// TIA Portal V17 export
// export: Created 2025-03-10T13:11:40.6014181Z, ExportSetting WithDefaults, DisplayName Totally Integrated Automation Portal, DisplayVersion V17 Update 8, DisplayName TIA Portal Openness, DisplayVersion V17 Update 8, DisplayName TIA Portal Version Control Interface, DisplayVersion V17, DisplayName SINAMICS Startdrive Advanced, DisplayVersion V17 SP2, DisplayName SINAMICS Startdrive G110M, G120, G120C, G120D, G120P, G115D, DisplayVersion V17 SP2, DisplayName SINAMICS Startdrive G130, G150, S120, S150, SINAMICS MV, S210, DisplayVersion V17 SP2, DisplayName STEP 7 Professional, DisplayVersion V17 Update 8, DisplayName SINUMERIK ONE STEP 7 Toolbox, DisplayVersion V17 Update 12, DisplayName SINUMERIK 840D sl STEP 7 Toolbox, DisplayVersion V17 Update 12, DisplayName STEP 7 Safety, DisplayVersion V17 Update 6, DisplayName WinCC Advanced, DisplayVersion V17 Update 8
FUNCTION "FC7213_CYCLE_TIMES_CLADDING" : Void   // FC7213, LAD
TITLE = FC CYCLE TIMES
{ S7_Optimized_Access := 'FALSE' }
AUTHOR : ETXETAR
VERSION : 1.0
// stored: AutoNumber false, IsIECCheckEnabled false, SetENOAutomatically false, UDAEnableTagReadback false
   VAR_TEMP
      CYCLE_TIME : Int;
      TIMER_INT : Int;
      PART_CYCLE_TIME : Int;
   END_VAR
   VAR_TEMP   // added for the SCL form of the ladder/FBD networks
      _w1 : Bool;
      _w2 : Bool;
      _w3 : Bool;
      _w4 : Bool;
   END_VAR
BEGIN

REGION Network 1: PART TYPE 1 TO 5
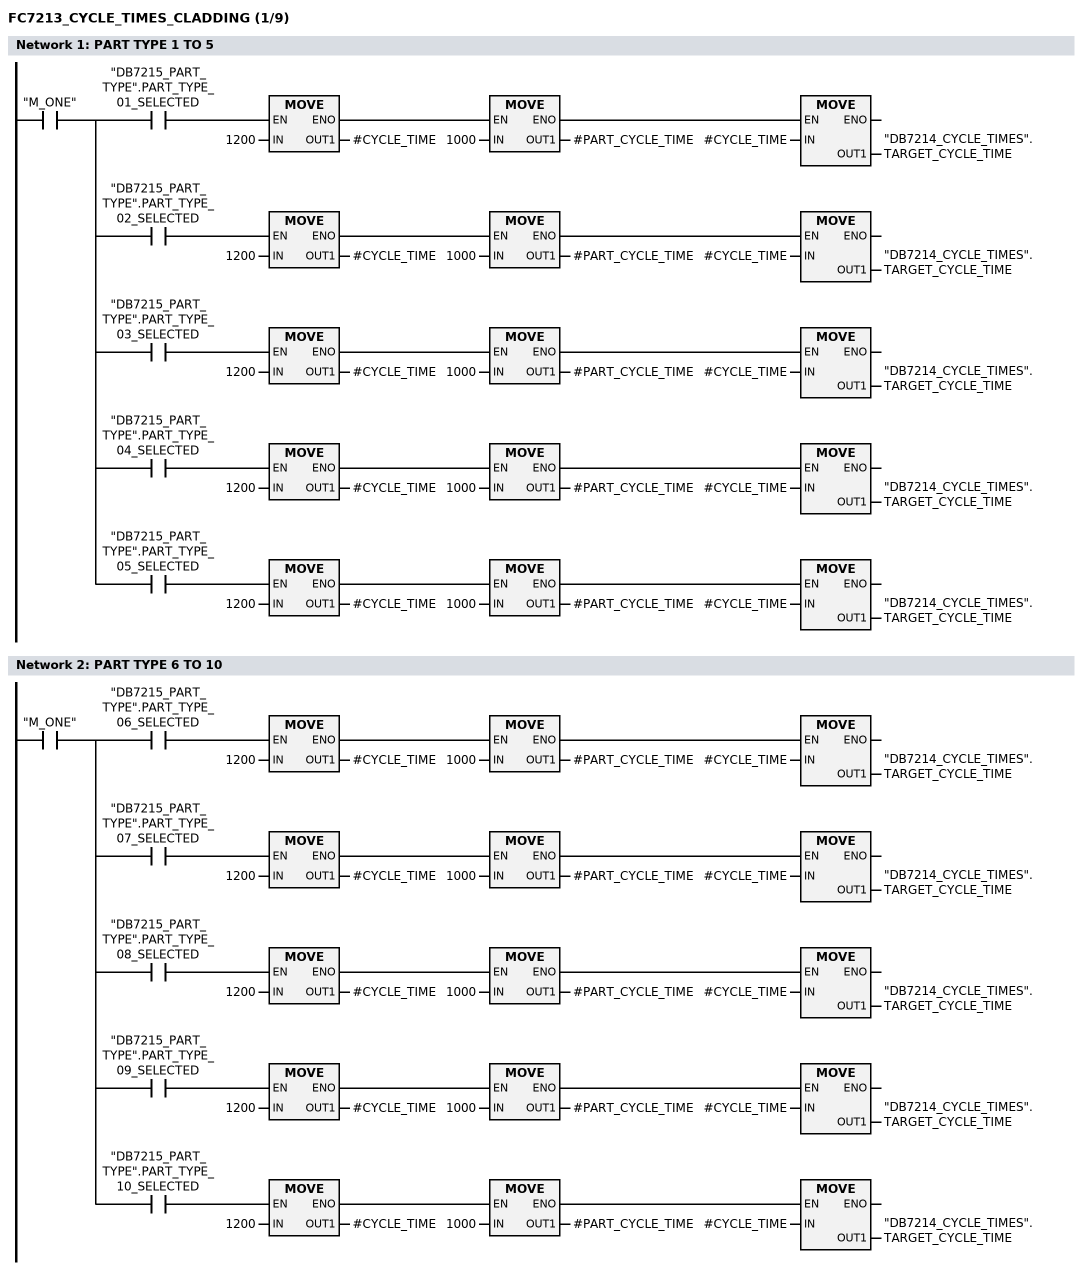
   RUNG wire#powerrail
      Contact( "M_ONE" )
      wire#w1
      Contact( "DB7215_PART_TYPE".PART_TYPE_01_SELECTED )
      { S7_GenerateENO := "TRUE" } Move(in := 1200, out1 => #CYCLE_TIME)
      { S7_GenerateENO := "TRUE" } Move(in := 1000, out1 => #PART_CYCLE_TIME)
      { S7_GenerateENO := "TRUE" } Move(in := #CYCLE_TIME, out1 => "DB7214_CYCLE_TIMES".TARGET_CYCLE_TIME)
   END_RUNG
   RUNG wire#w1
      Contact( "DB7215_PART_TYPE".PART_TYPE_02_SELECTED )
      { S7_GenerateENO := "TRUE" } Move(in := 1200, out1 => #CYCLE_TIME)
      { S7_GenerateENO := "TRUE" } Move(in := 1000, out1 => #PART_CYCLE_TIME)
      { S7_GenerateENO := "TRUE" } Move(in := #CYCLE_TIME, out1 => "DB7214_CYCLE_TIMES".TARGET_CYCLE_TIME)
   END_RUNG
   RUNG wire#w1
      Contact( "DB7215_PART_TYPE".PART_TYPE_03_SELECTED )
      { S7_GenerateENO := "TRUE" } Move(in := 1200, out1 => #CYCLE_TIME)
      { S7_GenerateENO := "TRUE" } Move(in := 1000, out1 => #PART_CYCLE_TIME)
      { S7_GenerateENO := "TRUE" } Move(in := #CYCLE_TIME, out1 => "DB7214_CYCLE_TIMES".TARGET_CYCLE_TIME)
   END_RUNG
   RUNG wire#w1
      Contact( "DB7215_PART_TYPE".PART_TYPE_04_SELECTED )
      { S7_GenerateENO := "TRUE" } Move(in := 1200, out1 => #CYCLE_TIME)
      { S7_GenerateENO := "TRUE" } Move(in := 1000, out1 => #PART_CYCLE_TIME)
      { S7_GenerateENO := "TRUE" } Move(in := #CYCLE_TIME, out1 => "DB7214_CYCLE_TIMES".TARGET_CYCLE_TIME)
   END_RUNG
   RUNG wire#w1
      Contact( "DB7215_PART_TYPE".PART_TYPE_05_SELECTED )
      { S7_GenerateENO := "TRUE" } Move(in := 1200, out1 => #CYCLE_TIME)
      { S7_GenerateENO := "TRUE" } Move(in := 1000, out1 => #PART_CYCLE_TIME)
      { S7_GenerateENO := "TRUE" } Move(in := #CYCLE_TIME, out1 => "DB7214_CYCLE_TIMES".TARGET_CYCLE_TIME)
   END_RUNG
   // the same network as SCL:
   // ENO of a box is taken as its EN; it also drops when the box reports an error
   IF "M_ONE" AND "DB7215_PART_TYPE".PART_TYPE_01_SELECTED THEN
       #CYCLE_TIME := 1200;
       #PART_CYCLE_TIME := 1000;
       "DB7214_CYCLE_TIMES".TARGET_CYCLE_TIME := #CYCLE_TIME;
   END_IF;
   IF "M_ONE" AND "DB7215_PART_TYPE".PART_TYPE_02_SELECTED THEN
       #CYCLE_TIME := 1200;
       #PART_CYCLE_TIME := 1000;
       "DB7214_CYCLE_TIMES".TARGET_CYCLE_TIME := #CYCLE_TIME;
   END_IF;
   IF "M_ONE" AND "DB7215_PART_TYPE".PART_TYPE_03_SELECTED THEN
       #CYCLE_TIME := 1200;
       #PART_CYCLE_TIME := 1000;
       "DB7214_CYCLE_TIMES".TARGET_CYCLE_TIME := #CYCLE_TIME;
   END_IF;
   IF "M_ONE" AND "DB7215_PART_TYPE".PART_TYPE_04_SELECTED THEN
       #CYCLE_TIME := 1200;
       #PART_CYCLE_TIME := 1000;
       "DB7214_CYCLE_TIMES".TARGET_CYCLE_TIME := #CYCLE_TIME;
   END_IF;
   IF "M_ONE" AND "DB7215_PART_TYPE".PART_TYPE_05_SELECTED THEN
       #CYCLE_TIME := 1200;
       #PART_CYCLE_TIME := 1000;
       "DB7214_CYCLE_TIMES".TARGET_CYCLE_TIME := #CYCLE_TIME;
   END_IF;
END_REGION

REGION Network 2: PART TYPE 6 TO 10
   RUNG wire#powerrail
      Contact( "M_ONE" )
      wire#w1
      Contact( "DB7215_PART_TYPE".PART_TYPE_06_SELECTED )
      { S7_GenerateENO := "TRUE" } Move(in := 1200, out1 => #CYCLE_TIME)
      { S7_GenerateENO := "TRUE" } Move(in := 1000, out1 => #PART_CYCLE_TIME)
      { S7_GenerateENO := "TRUE" } Move(in := #CYCLE_TIME, out1 => "DB7214_CYCLE_TIMES".TARGET_CYCLE_TIME)
   END_RUNG
   RUNG wire#w1
      Contact( "DB7215_PART_TYPE".PART_TYPE_07_SELECTED )
      { S7_GenerateENO := "TRUE" } Move(in := 1200, out1 => #CYCLE_TIME)
      { S7_GenerateENO := "TRUE" } Move(in := 1000, out1 => #PART_CYCLE_TIME)
      { S7_GenerateENO := "TRUE" } Move(in := #CYCLE_TIME, out1 => "DB7214_CYCLE_TIMES".TARGET_CYCLE_TIME)
   END_RUNG
   RUNG wire#w1
      Contact( "DB7215_PART_TYPE".PART_TYPE_08_SELECTED )
      { S7_GenerateENO := "TRUE" } Move(in := 1200, out1 => #CYCLE_TIME)
      { S7_GenerateENO := "TRUE" } Move(in := 1000, out1 => #PART_CYCLE_TIME)
      { S7_GenerateENO := "TRUE" } Move(in := #CYCLE_TIME, out1 => "DB7214_CYCLE_TIMES".TARGET_CYCLE_TIME)
   END_RUNG
   RUNG wire#w1
      Contact( "DB7215_PART_TYPE".PART_TYPE_09_SELECTED )
      { S7_GenerateENO := "TRUE" } Move(in := 1200, out1 => #CYCLE_TIME)
      { S7_GenerateENO := "TRUE" } Move(in := 1000, out1 => #PART_CYCLE_TIME)
      { S7_GenerateENO := "TRUE" } Move(in := #CYCLE_TIME, out1 => "DB7214_CYCLE_TIMES".TARGET_CYCLE_TIME)
   END_RUNG
   RUNG wire#w1
      Contact( "DB7215_PART_TYPE".PART_TYPE_10_SELECTED )
      { S7_GenerateENO := "TRUE" } Move(in := 1200, out1 => #CYCLE_TIME)
      { S7_GenerateENO := "TRUE" } Move(in := 1000, out1 => #PART_CYCLE_TIME)
      { S7_GenerateENO := "TRUE" } Move(in := #CYCLE_TIME, out1 => "DB7214_CYCLE_TIMES".TARGET_CYCLE_TIME)
   END_RUNG
   // the same network as SCL:
   // ENO of a box is taken as its EN; it also drops when the box reports an error
   IF "M_ONE" AND "DB7215_PART_TYPE".PART_TYPE_06_SELECTED THEN
       #CYCLE_TIME := 1200;
       #PART_CYCLE_TIME := 1000;
       "DB7214_CYCLE_TIMES".TARGET_CYCLE_TIME := #CYCLE_TIME;
   END_IF;
   IF "M_ONE" AND "DB7215_PART_TYPE".PART_TYPE_07_SELECTED THEN
       #CYCLE_TIME := 1200;
       #PART_CYCLE_TIME := 1000;
       "DB7214_CYCLE_TIMES".TARGET_CYCLE_TIME := #CYCLE_TIME;
   END_IF;
   IF "M_ONE" AND "DB7215_PART_TYPE".PART_TYPE_08_SELECTED THEN
       #CYCLE_TIME := 1200;
       #PART_CYCLE_TIME := 1000;
       "DB7214_CYCLE_TIMES".TARGET_CYCLE_TIME := #CYCLE_TIME;
   END_IF;
   IF "M_ONE" AND "DB7215_PART_TYPE".PART_TYPE_09_SELECTED THEN
       #CYCLE_TIME := 1200;
       #PART_CYCLE_TIME := 1000;
       "DB7214_CYCLE_TIMES".TARGET_CYCLE_TIME := #CYCLE_TIME;
   END_IF;
   IF "M_ONE" AND "DB7215_PART_TYPE".PART_TYPE_10_SELECTED THEN
       #CYCLE_TIME := 1200;
       #PART_CYCLE_TIME := 1000;
       "DB7214_CYCLE_TIMES".TARGET_CYCLE_TIME := #CYCLE_TIME;
   END_IF;
END_REGION

REGION Network 3: PART TYPE 11 TO 15
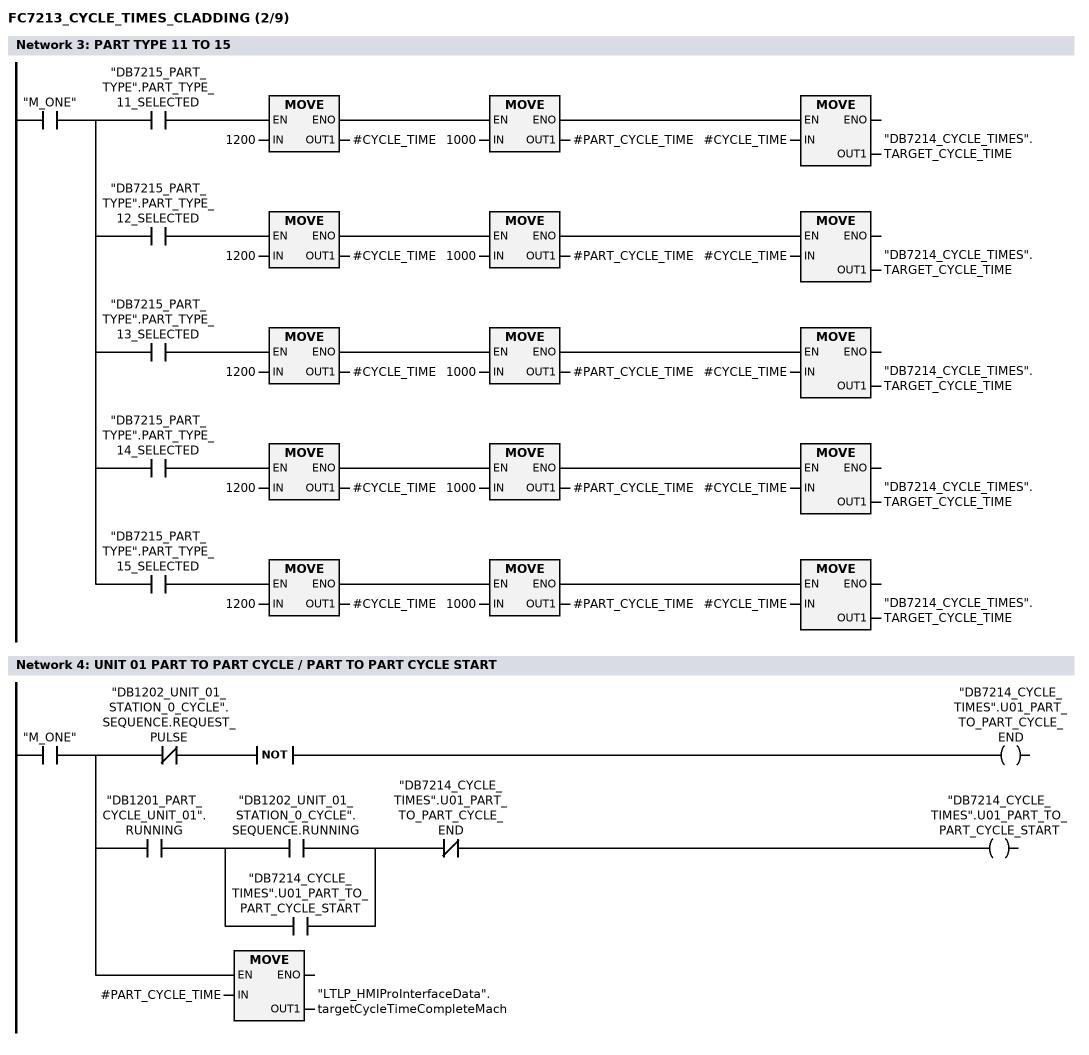
   RUNG wire#powerrail
      Contact( "M_ONE" )
      wire#w1
      Contact( "DB7215_PART_TYPE".PART_TYPE_11_SELECTED )
      { S7_GenerateENO := "TRUE" } Move(in := 1200, out1 => #CYCLE_TIME)
      { S7_GenerateENO := "TRUE" } Move(in := 1000, out1 => #PART_CYCLE_TIME)
      { S7_GenerateENO := "TRUE" } Move(in := #CYCLE_TIME, out1 => "DB7214_CYCLE_TIMES".TARGET_CYCLE_TIME)
   END_RUNG
   RUNG wire#w1
      Contact( "DB7215_PART_TYPE".PART_TYPE_12_SELECTED )
      { S7_GenerateENO := "TRUE" } Move(in := 1200, out1 => #CYCLE_TIME)
      { S7_GenerateENO := "TRUE" } Move(in := 1000, out1 => #PART_CYCLE_TIME)
      { S7_GenerateENO := "TRUE" } Move(in := #CYCLE_TIME, out1 => "DB7214_CYCLE_TIMES".TARGET_CYCLE_TIME)
   END_RUNG
   RUNG wire#w1
      Contact( "DB7215_PART_TYPE".PART_TYPE_13_SELECTED )
      { S7_GenerateENO := "TRUE" } Move(in := 1200, out1 => #CYCLE_TIME)
      { S7_GenerateENO := "TRUE" } Move(in := 1000, out1 => #PART_CYCLE_TIME)
      { S7_GenerateENO := "TRUE" } Move(in := #CYCLE_TIME, out1 => "DB7214_CYCLE_TIMES".TARGET_CYCLE_TIME)
   END_RUNG
   RUNG wire#w1
      Contact( "DB7215_PART_TYPE".PART_TYPE_14_SELECTED )
      { S7_GenerateENO := "TRUE" } Move(in := 1200, out1 => #CYCLE_TIME)
      { S7_GenerateENO := "TRUE" } Move(in := 1000, out1 => #PART_CYCLE_TIME)
      { S7_GenerateENO := "TRUE" } Move(in := #CYCLE_TIME, out1 => "DB7214_CYCLE_TIMES".TARGET_CYCLE_TIME)
   END_RUNG
   RUNG wire#w1
      Contact( "DB7215_PART_TYPE".PART_TYPE_15_SELECTED )
      { S7_GenerateENO := "TRUE" } Move(in := 1200, out1 => #CYCLE_TIME)
      { S7_GenerateENO := "TRUE" } Move(in := 1000, out1 => #PART_CYCLE_TIME)
      { S7_GenerateENO := "TRUE" } Move(in := #CYCLE_TIME, out1 => "DB7214_CYCLE_TIMES".TARGET_CYCLE_TIME)
   END_RUNG
   // the same network as SCL:
   // ENO of a box is taken as its EN; it also drops when the box reports an error
   IF "M_ONE" AND "DB7215_PART_TYPE".PART_TYPE_11_SELECTED THEN
       #CYCLE_TIME := 1200;
       #PART_CYCLE_TIME := 1000;
       "DB7214_CYCLE_TIMES".TARGET_CYCLE_TIME := #CYCLE_TIME;
   END_IF;
   IF "M_ONE" AND "DB7215_PART_TYPE".PART_TYPE_12_SELECTED THEN
       #CYCLE_TIME := 1200;
       #PART_CYCLE_TIME := 1000;
       "DB7214_CYCLE_TIMES".TARGET_CYCLE_TIME := #CYCLE_TIME;
   END_IF;
   IF "M_ONE" AND "DB7215_PART_TYPE".PART_TYPE_13_SELECTED THEN
       #CYCLE_TIME := 1200;
       #PART_CYCLE_TIME := 1000;
       "DB7214_CYCLE_TIMES".TARGET_CYCLE_TIME := #CYCLE_TIME;
   END_IF;
   IF "M_ONE" AND "DB7215_PART_TYPE".PART_TYPE_14_SELECTED THEN
       #CYCLE_TIME := 1200;
       #PART_CYCLE_TIME := 1000;
       "DB7214_CYCLE_TIMES".TARGET_CYCLE_TIME := #CYCLE_TIME;
   END_IF;
   IF "M_ONE" AND "DB7215_PART_TYPE".PART_TYPE_15_SELECTED THEN
       #CYCLE_TIME := 1200;
       #PART_CYCLE_TIME := 1000;
       "DB7214_CYCLE_TIMES".TARGET_CYCLE_TIME := #CYCLE_TIME;
   END_IF;
END_REGION

REGION Network 4: UNIT 01 PART TO PART CYCLE / PART TO PART CYCLE START
   RUNG wire#powerrail
      Contact( "M_ONE" )
      wire#w1
      I_Contact( "DB1202_UNIT_01_STATION_0_CYCLE".SEQUENCE.REQUEST_PULSE )
      Not()
      Coil( "DB7214_CYCLE_TIMES".U01_PART_TO_PART_CYCLE_END )
   END_RUNG
   RUNG wire#w1
      Contact( "DB1201_PART_CYCLE_UNIT_01".RUNNING )
      wire#w2
      Contact( "DB1202_UNIT_01_STATION_0_CYCLE".SEQUENCE.RUNNING )
      wire#w3
      I_Contact( "DB7214_CYCLE_TIMES".U01_PART_TO_PART_CYCLE_END )
      Coil( "DB7214_CYCLE_TIMES".U01_PART_TO_PART_CYCLE_START )
   END_RUNG
   RUNG wire#w2
      Contact( "DB7214_CYCLE_TIMES".U01_PART_TO_PART_CYCLE_START )
   END_RUNG wire#w3
   RUNG wire#w1
      { S7_GenerateENO := "TRUE" } Move(in := #PART_CYCLE_TIME, out1 => "LTLP_HMIProInterfaceData".targetCycleTimeCompleteMach)
   END_RUNG
   // the same network as SCL:
   "DB7214_CYCLE_TIMES".U01_PART_TO_PART_CYCLE_END := NOT ("M_ONE" AND NOT "DB1202_UNIT_01_STATION_0_CYCLE".SEQUENCE.REQUEST_PULSE);
   "DB7214_CYCLE_TIMES".U01_PART_TO_PART_CYCLE_START := "M_ONE" AND "DB1201_PART_CYCLE_UNIT_01".RUNNING AND ("DB1202_UNIT_01_STATION_0_CYCLE".SEQUENCE.RUNNING OR "DB7214_CYCLE_TIMES".U01_PART_TO_PART_CYCLE_START) AND NOT "DB7214_CYCLE_TIMES".U01_PART_TO_PART_CYCLE_END;
   IF "M_ONE" THEN "LTLP_HMIProInterfaceData".targetCycleTimeCompleteMach := #PART_CYCLE_TIME; END_IF;
END_REGION

NETWORK
TITLE = UNIT 01 HMI HISTORY
      L     "LTLP_HMIProInterfaceData".targetCycleTimeCompleteMach;
      T     "LTLP_HMIProInterfaceData".targetCycleTime[13];
      T     "LTLP_HMIProInterfaceData".targetCycleTime[14];
      T     "LTLP_HMIProInterfaceData".targetCycleTime[15];
      T     "LTLP_HMIProInterfaceData".targetCycleTime[16];
      T     "LTLP_HMIProInterfaceData".targetCycleTime[17];
      T     "LTLP_HMIProInterfaceData".targetCycleTime[18];
      T     "LTLP_HMIProInterfaceData".targetCycleTime[19];
      T     "LTLP_HMIProInterfaceData".targetCycleTime[20];
      T     "LTLP_HMIProInterfaceData".targetCycleTime[21];
      T     "LTLP_HMIProInterfaceData".targetCycleTime[22];
      NOP   0;

REGION Network 6: UNIT 01 MOVE HMI HISTORY
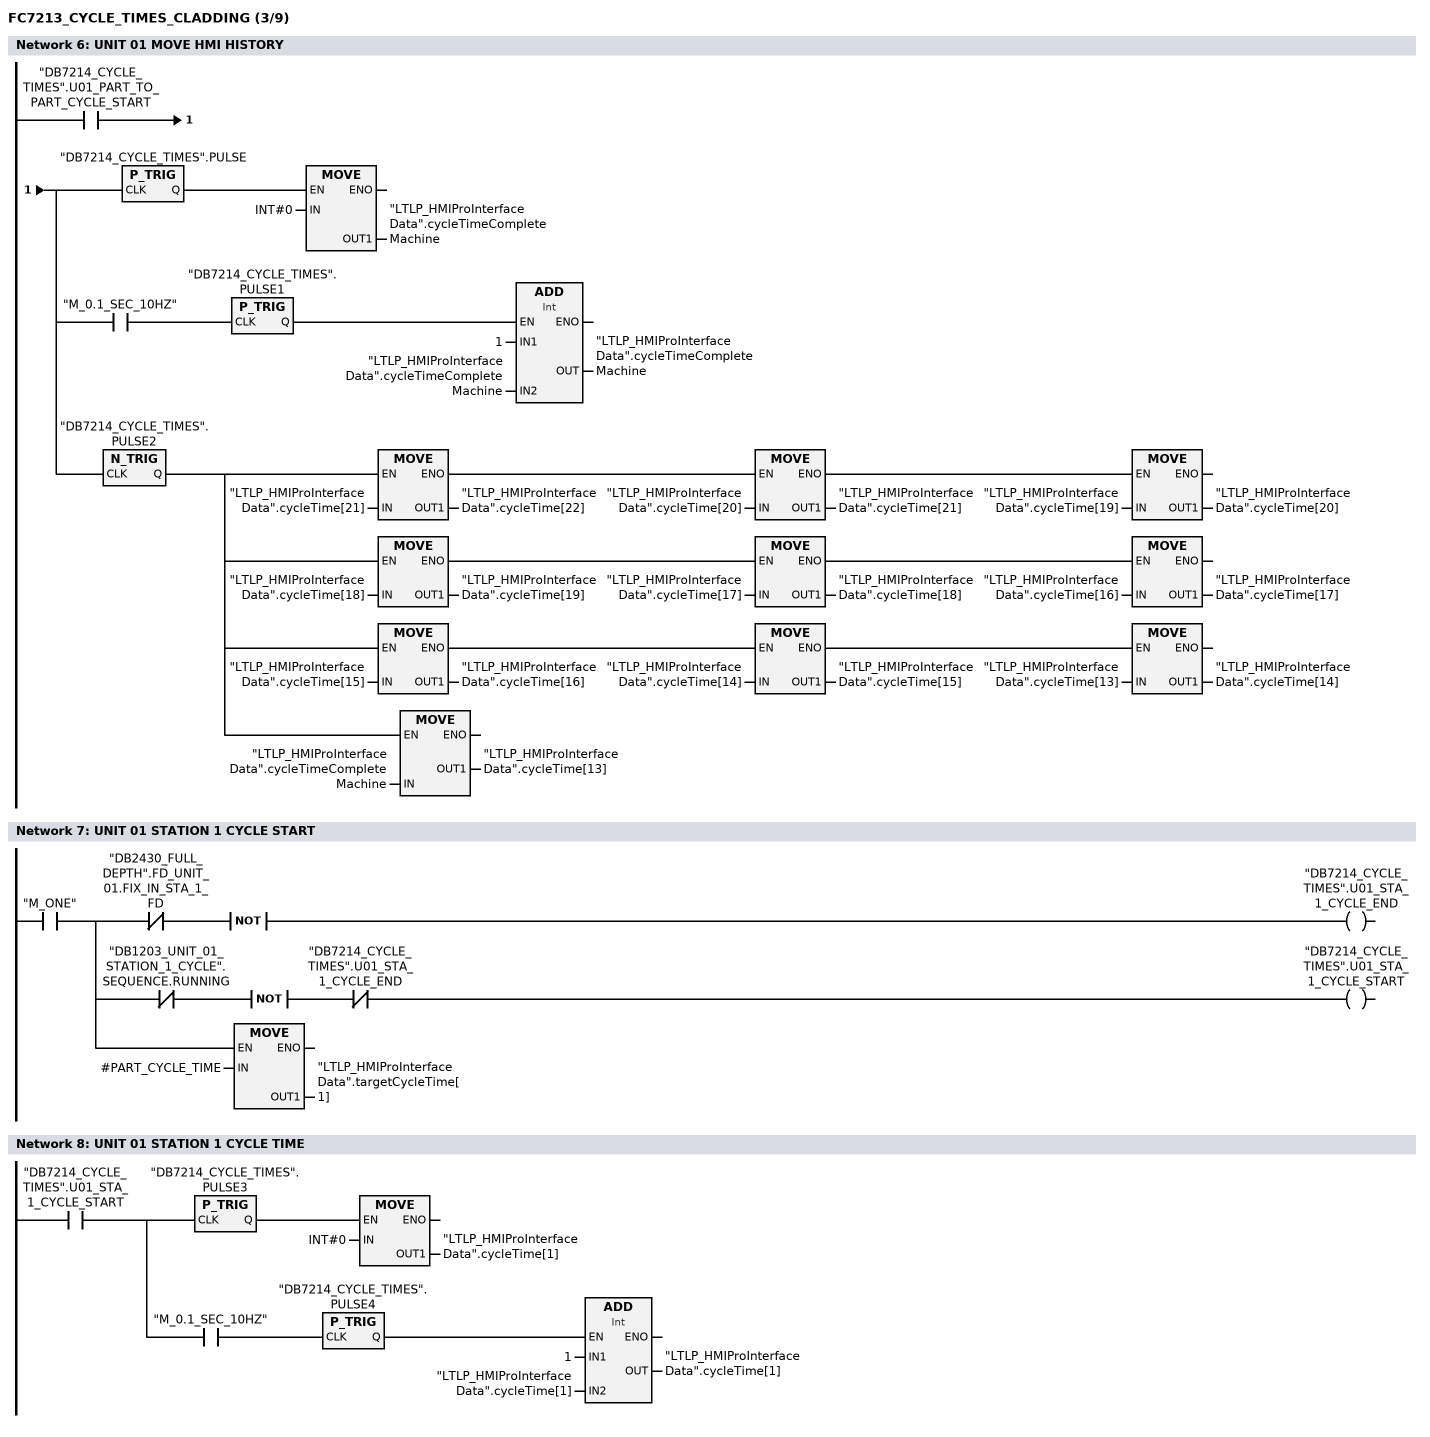
   RUNG wire#powerrail
      Contact( "DB7214_CYCLE_TIMES".U01_PART_TO_PART_CYCLE_START )
      wire#w1
      P_Trig( "DB7214_CYCLE_TIMES".PULSE )
      { S7_GenerateENO := "TRUE" } Move(in := INT#0, out1 => "LTLP_HMIProInterfaceData".cycleTimeCompleteMachine)
   END_RUNG
   RUNG wire#w1
      Contact( "M_0.1_SEC_10HZ" )
      P_Trig( "DB7214_CYCLE_TIMES".PULSE1 )
      { S7_Templates := "SrcType := Int"; S7_GenerateENO := "TRUE" } Add(in1 := 1, in2 := "LTLP_HMIProInterfaceData".cycleTimeCompleteMachine, out => "LTLP_HMIProInterfaceData".cycleTimeCompleteMachine)
   END_RUNG
   RUNG wire#w1
      N_Trig( "DB7214_CYCLE_TIMES".PULSE2 )
      wire#w2
      { S7_GenerateENO := "TRUE" } Move(in := "LTLP_HMIProInterfaceData".cycleTime[21], out1 => "LTLP_HMIProInterfaceData".cycleTime[22])
      { S7_GenerateENO := "TRUE" } Move(in := "LTLP_HMIProInterfaceData".cycleTime[20], out1 => "LTLP_HMIProInterfaceData".cycleTime[21])
      { S7_GenerateENO := "TRUE" } Move(in := "LTLP_HMIProInterfaceData".cycleTime[19], out1 => "LTLP_HMIProInterfaceData".cycleTime[20])
   END_RUNG
   RUNG wire#w2
      { S7_GenerateENO := "TRUE" } Move(in := "LTLP_HMIProInterfaceData".cycleTime[18], out1 => "LTLP_HMIProInterfaceData".cycleTime[19])
      { S7_GenerateENO := "TRUE" } Move(in := "LTLP_HMIProInterfaceData".cycleTime[17], out1 => "LTLP_HMIProInterfaceData".cycleTime[18])
      { S7_GenerateENO := "TRUE" } Move(in := "LTLP_HMIProInterfaceData".cycleTime[16], out1 => "LTLP_HMIProInterfaceData".cycleTime[17])
   END_RUNG
   RUNG wire#w2
      { S7_GenerateENO := "TRUE" } Move(in := "LTLP_HMIProInterfaceData".cycleTime[15], out1 => "LTLP_HMIProInterfaceData".cycleTime[16])
      { S7_GenerateENO := "TRUE" } Move(in := "LTLP_HMIProInterfaceData".cycleTime[14], out1 => "LTLP_HMIProInterfaceData".cycleTime[15])
      { S7_GenerateENO := "TRUE" } Move(in := "LTLP_HMIProInterfaceData".cycleTime[13], out1 => "LTLP_HMIProInterfaceData".cycleTime[14])
   END_RUNG
   RUNG wire#w2
      { S7_GenerateENO := "TRUE" } Move(in := "LTLP_HMIProInterfaceData".cycleTimeCompleteMachine, out1 => "LTLP_HMIProInterfaceData".cycleTime[13])
   END_RUNG
   // the same network as SCL:
   // ENO of a box is taken as its EN; it also drops when the box reports an error
   #_w1 := "DB7214_CYCLE_TIMES".U01_PART_TO_PART_CYCLE_START AND NOT "DB7214_CYCLE_TIMES".PULSE;   // rising edge
   "DB7214_CYCLE_TIMES".PULSE := "DB7214_CYCLE_TIMES".U01_PART_TO_PART_CYCLE_START;
   IF #_w1 THEN "LTLP_HMIProInterfaceData".cycleTimeCompleteMachine := INT#0; END_IF;
   #_w2 := "DB7214_CYCLE_TIMES".U01_PART_TO_PART_CYCLE_START AND "M_0.1_SEC_10HZ";
   #_w3 := #_w2 AND NOT "DB7214_CYCLE_TIMES".PULSE1;   // rising edge
   "DB7214_CYCLE_TIMES".PULSE1 := #_w2;
   IF #_w3 THEN
       "LTLP_HMIProInterfaceData".cycleTimeCompleteMachine := 1 + "LTLP_HMIProInterfaceData".cycleTimeCompleteMachine;
   END_IF;
   #_w4 := NOT "DB7214_CYCLE_TIMES".U01_PART_TO_PART_CYCLE_START AND "DB7214_CYCLE_TIMES".PULSE2;   // falling edge
   "DB7214_CYCLE_TIMES".PULSE2 := "DB7214_CYCLE_TIMES".U01_PART_TO_PART_CYCLE_START;
   IF #_w4 THEN
       "LTLP_HMIProInterfaceData".cycleTime[22] := "LTLP_HMIProInterfaceData".cycleTime[21];
       "LTLP_HMIProInterfaceData".cycleTime[21] := "LTLP_HMIProInterfaceData".cycleTime[20];
       "LTLP_HMIProInterfaceData".cycleTime[20] := "LTLP_HMIProInterfaceData".cycleTime[19];
       "LTLP_HMIProInterfaceData".cycleTime[19] := "LTLP_HMIProInterfaceData".cycleTime[18];
       "LTLP_HMIProInterfaceData".cycleTime[18] := "LTLP_HMIProInterfaceData".cycleTime[17];
       "LTLP_HMIProInterfaceData".cycleTime[17] := "LTLP_HMIProInterfaceData".cycleTime[16];
       "LTLP_HMIProInterfaceData".cycleTime[16] := "LTLP_HMIProInterfaceData".cycleTime[15];
       "LTLP_HMIProInterfaceData".cycleTime[15] := "LTLP_HMIProInterfaceData".cycleTime[14];
       "LTLP_HMIProInterfaceData".cycleTime[14] := "LTLP_HMIProInterfaceData".cycleTime[13];
       "LTLP_HMIProInterfaceData".cycleTime[13] := "LTLP_HMIProInterfaceData".cycleTimeCompleteMachine;
   END_IF;
END_REGION

REGION Network 7: UNIT 01 STATION 1 CYCLE START
   RUNG wire#powerrail
      Contact( "M_ONE" )
      wire#w1
      I_Contact( "DB2430_FULL_DEPTH".FD_UNIT_01.FIX_IN_STA_1_FD )
      Not()
      Coil( "DB7214_CYCLE_TIMES".U01_STA_1_CYCLE_END )
   END_RUNG
   RUNG wire#w1
      I_Contact( "DB1203_UNIT_01_STATION_1_CYCLE".SEQUENCE.RUNNING )
      Not()
      I_Contact( "DB7214_CYCLE_TIMES".U01_STA_1_CYCLE_END )
      Coil( "DB7214_CYCLE_TIMES".U01_STA_1_CYCLE_START )
   END_RUNG
   RUNG wire#w1
      { S7_GenerateENO := "TRUE" } Move(in := #PART_CYCLE_TIME, out1 => "LTLP_HMIProInterfaceData".targetCycleTime[1])
   END_RUNG
   // the same network as SCL:
   "DB7214_CYCLE_TIMES".U01_STA_1_CYCLE_END := NOT ("M_ONE" AND NOT "DB2430_FULL_DEPTH".FD_UNIT_01.FIX_IN_STA_1_FD);
   "DB7214_CYCLE_TIMES".U01_STA_1_CYCLE_START := NOT ("M_ONE" AND NOT "DB1203_UNIT_01_STATION_1_CYCLE".SEQUENCE.RUNNING) AND NOT "DB7214_CYCLE_TIMES".U01_STA_1_CYCLE_END;
   IF "M_ONE" THEN "LTLP_HMIProInterfaceData".targetCycleTime[1] := #PART_CYCLE_TIME; END_IF;
END_REGION

REGION Network 8: UNIT 01 STATION 1 CYCLE TIME
   RUNG wire#powerrail
      Contact( "DB7214_CYCLE_TIMES".U01_STA_1_CYCLE_START )
      wire#w1
      P_Trig( "DB7214_CYCLE_TIMES".PULSE3 )
      { S7_GenerateENO := "TRUE" } Move(in := INT#0, out1 => "LTLP_HMIProInterfaceData".cycleTime[1])
   END_RUNG
   RUNG wire#w1
      Contact( "M_0.1_SEC_10HZ" )
      P_Trig( "DB7214_CYCLE_TIMES".PULSE4 )
      { S7_Templates := "SrcType := Int"; S7_GenerateENO := "TRUE" } Add(in1 := 1, in2 := "LTLP_HMIProInterfaceData".cycleTime[1], out => "LTLP_HMIProInterfaceData".cycleTime[1])
   END_RUNG
   // the same network as SCL:
   #_w1 := "DB7214_CYCLE_TIMES".U01_STA_1_CYCLE_START AND NOT "DB7214_CYCLE_TIMES".PULSE3;   // rising edge
   "DB7214_CYCLE_TIMES".PULSE3 := "DB7214_CYCLE_TIMES".U01_STA_1_CYCLE_START;
   IF #_w1 THEN "LTLP_HMIProInterfaceData".cycleTime[1] := INT#0; END_IF;
   #_w2 := "DB7214_CYCLE_TIMES".U01_STA_1_CYCLE_START AND "M_0.1_SEC_10HZ";
   #_w3 := #_w2 AND NOT "DB7214_CYCLE_TIMES".PULSE4;   // rising edge
   "DB7214_CYCLE_TIMES".PULSE4 := #_w2;
   IF #_w3 THEN
       "LTLP_HMIProInterfaceData".cycleTime[1] := 1 + "LTLP_HMIProInterfaceData".cycleTime[1];
   END_IF;
END_REGION

REGION Network 9: UNIT 01 STATION 2 CYCLE START
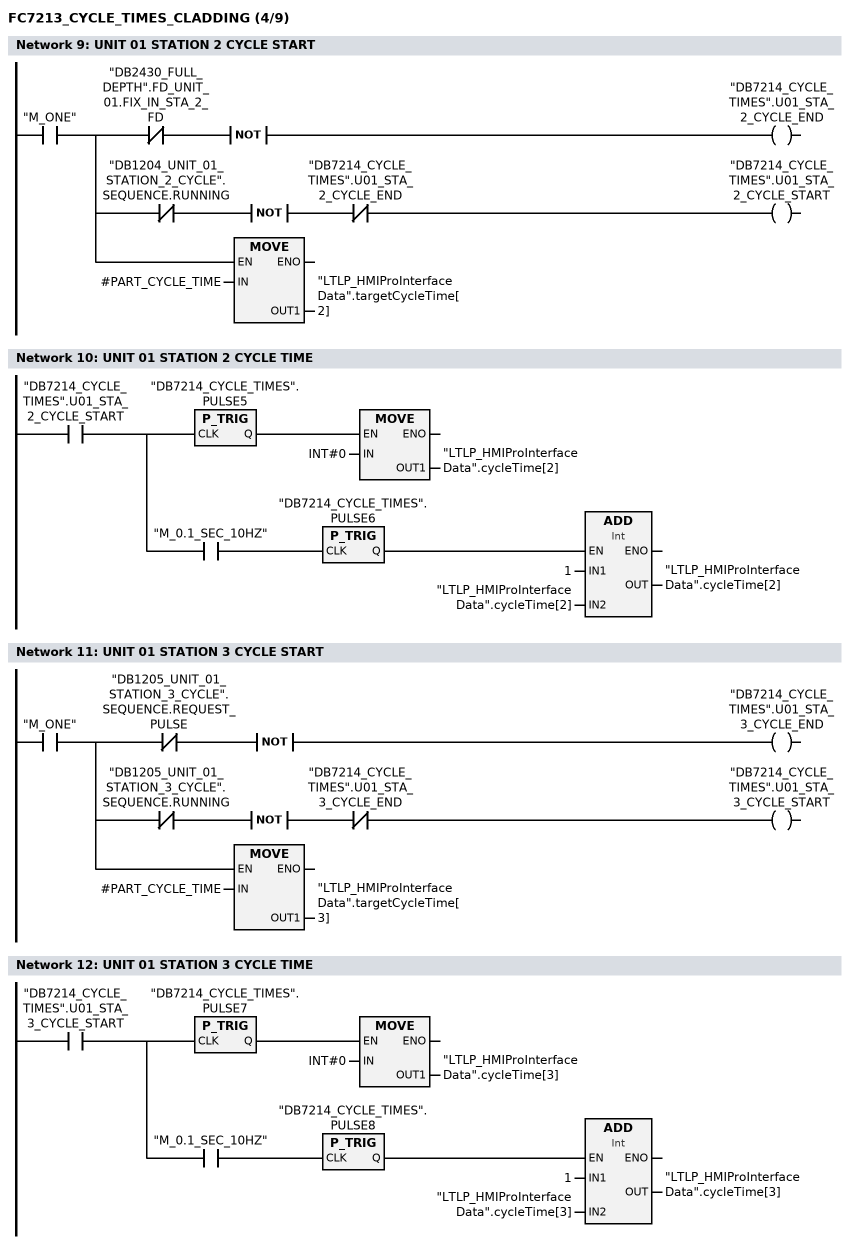
   RUNG wire#powerrail
      Contact( "M_ONE" )
      wire#w1
      I_Contact( "DB2430_FULL_DEPTH".FD_UNIT_01.FIX_IN_STA_2_FD )
      Not()
      Coil( "DB7214_CYCLE_TIMES".U01_STA_2_CYCLE_END )
   END_RUNG
   RUNG wire#w1
      I_Contact( "DB1204_UNIT_01_STATION_2_CYCLE".SEQUENCE.RUNNING )
      Not()
      I_Contact( "DB7214_CYCLE_TIMES".U01_STA_2_CYCLE_END )
      Coil( "DB7214_CYCLE_TIMES".U01_STA_2_CYCLE_START )
   END_RUNG
   RUNG wire#w1
      { S7_GenerateENO := "TRUE" } Move(in := #PART_CYCLE_TIME, out1 => "LTLP_HMIProInterfaceData".targetCycleTime[2])
   END_RUNG
   // the same network as SCL:
   "DB7214_CYCLE_TIMES".U01_STA_2_CYCLE_END := NOT ("M_ONE" AND NOT "DB2430_FULL_DEPTH".FD_UNIT_01.FIX_IN_STA_2_FD);
   "DB7214_CYCLE_TIMES".U01_STA_2_CYCLE_START := NOT ("M_ONE" AND NOT "DB1204_UNIT_01_STATION_2_CYCLE".SEQUENCE.RUNNING) AND NOT "DB7214_CYCLE_TIMES".U01_STA_2_CYCLE_END;
   IF "M_ONE" THEN "LTLP_HMIProInterfaceData".targetCycleTime[2] := #PART_CYCLE_TIME; END_IF;
END_REGION

REGION Network 10: UNIT 01 STATION 2 CYCLE TIME
   RUNG wire#powerrail
      Contact( "DB7214_CYCLE_TIMES".U01_STA_2_CYCLE_START )
      wire#w1
      P_Trig( "DB7214_CYCLE_TIMES".PULSE5 )
      { S7_GenerateENO := "TRUE" } Move(in := INT#0, out1 => "LTLP_HMIProInterfaceData".cycleTime[2])
   END_RUNG
   RUNG wire#w1
      Contact( "M_0.1_SEC_10HZ" )
      P_Trig( "DB7214_CYCLE_TIMES".PULSE6 )
      { S7_Templates := "SrcType := Int"; S7_GenerateENO := "TRUE" } Add(in1 := 1, in2 := "LTLP_HMIProInterfaceData".cycleTime[2], out => "LTLP_HMIProInterfaceData".cycleTime[2])
   END_RUNG
   // the same network as SCL:
   #_w1 := "DB7214_CYCLE_TIMES".U01_STA_2_CYCLE_START AND NOT "DB7214_CYCLE_TIMES".PULSE5;   // rising edge
   "DB7214_CYCLE_TIMES".PULSE5 := "DB7214_CYCLE_TIMES".U01_STA_2_CYCLE_START;
   IF #_w1 THEN "LTLP_HMIProInterfaceData".cycleTime[2] := INT#0; END_IF;
   #_w2 := "DB7214_CYCLE_TIMES".U01_STA_2_CYCLE_START AND "M_0.1_SEC_10HZ";
   #_w3 := #_w2 AND NOT "DB7214_CYCLE_TIMES".PULSE6;   // rising edge
   "DB7214_CYCLE_TIMES".PULSE6 := #_w2;
   IF #_w3 THEN
       "LTLP_HMIProInterfaceData".cycleTime[2] := 1 + "LTLP_HMIProInterfaceData".cycleTime[2];
   END_IF;
END_REGION

REGION Network 11: UNIT 01 STATION 3 CYCLE START
   RUNG wire#powerrail
      Contact( "M_ONE" )
      wire#w1
      I_Contact( "DB1205_UNIT_01_STATION_3_CYCLE".SEQUENCE.REQUEST_PULSE )
      Not()
      Coil( "DB7214_CYCLE_TIMES".U01_STA_3_CYCLE_END )
   END_RUNG
   RUNG wire#w1
      I_Contact( "DB1205_UNIT_01_STATION_3_CYCLE".SEQUENCE.RUNNING )
      Not()
      I_Contact( "DB7214_CYCLE_TIMES".U01_STA_3_CYCLE_END )
      Coil( "DB7214_CYCLE_TIMES".U01_STA_3_CYCLE_START )
   END_RUNG
   RUNG wire#w1
      { S7_GenerateENO := "TRUE" } Move(in := #PART_CYCLE_TIME, out1 => "LTLP_HMIProInterfaceData".targetCycleTime[3])
   END_RUNG
   // the same network as SCL:
   "DB7214_CYCLE_TIMES".U01_STA_3_CYCLE_END := NOT ("M_ONE" AND NOT "DB1205_UNIT_01_STATION_3_CYCLE".SEQUENCE.REQUEST_PULSE);
   "DB7214_CYCLE_TIMES".U01_STA_3_CYCLE_START := NOT ("M_ONE" AND NOT "DB1205_UNIT_01_STATION_3_CYCLE".SEQUENCE.RUNNING) AND NOT "DB7214_CYCLE_TIMES".U01_STA_3_CYCLE_END;
   IF "M_ONE" THEN "LTLP_HMIProInterfaceData".targetCycleTime[3] := #PART_CYCLE_TIME; END_IF;
END_REGION

REGION Network 12: UNIT 01 STATION 3 CYCLE TIME
   RUNG wire#powerrail
      Contact( "DB7214_CYCLE_TIMES".U01_STA_3_CYCLE_START )
      wire#w1
      P_Trig( "DB7214_CYCLE_TIMES".PULSE7 )
      { S7_GenerateENO := "TRUE" } Move(in := INT#0, out1 => "LTLP_HMIProInterfaceData".cycleTime[3])
   END_RUNG
   RUNG wire#w1
      Contact( "M_0.1_SEC_10HZ" )
      P_Trig( "DB7214_CYCLE_TIMES".PULSE8 )
      { S7_Templates := "SrcType := Int"; S7_GenerateENO := "TRUE" } Add(in1 := 1, in2 := "LTLP_HMIProInterfaceData".cycleTime[3], out => "LTLP_HMIProInterfaceData".cycleTime[3])
   END_RUNG
   // the same network as SCL:
   #_w1 := "DB7214_CYCLE_TIMES".U01_STA_3_CYCLE_START AND NOT "DB7214_CYCLE_TIMES".PULSE7;   // rising edge
   "DB7214_CYCLE_TIMES".PULSE7 := "DB7214_CYCLE_TIMES".U01_STA_3_CYCLE_START;
   IF #_w1 THEN "LTLP_HMIProInterfaceData".cycleTime[3] := INT#0; END_IF;
   #_w2 := "DB7214_CYCLE_TIMES".U01_STA_3_CYCLE_START AND "M_0.1_SEC_10HZ";
   #_w3 := #_w2 AND NOT "DB7214_CYCLE_TIMES".PULSE8;   // rising edge
   "DB7214_CYCLE_TIMES".PULSE8 := #_w2;
   IF #_w3 THEN
       "LTLP_HMIProInterfaceData".cycleTime[3] := 1 + "LTLP_HMIProInterfaceData".cycleTime[3];
   END_IF;
END_REGION

REGION Network 13: UNIT 01 STATION 4 CYCLE START
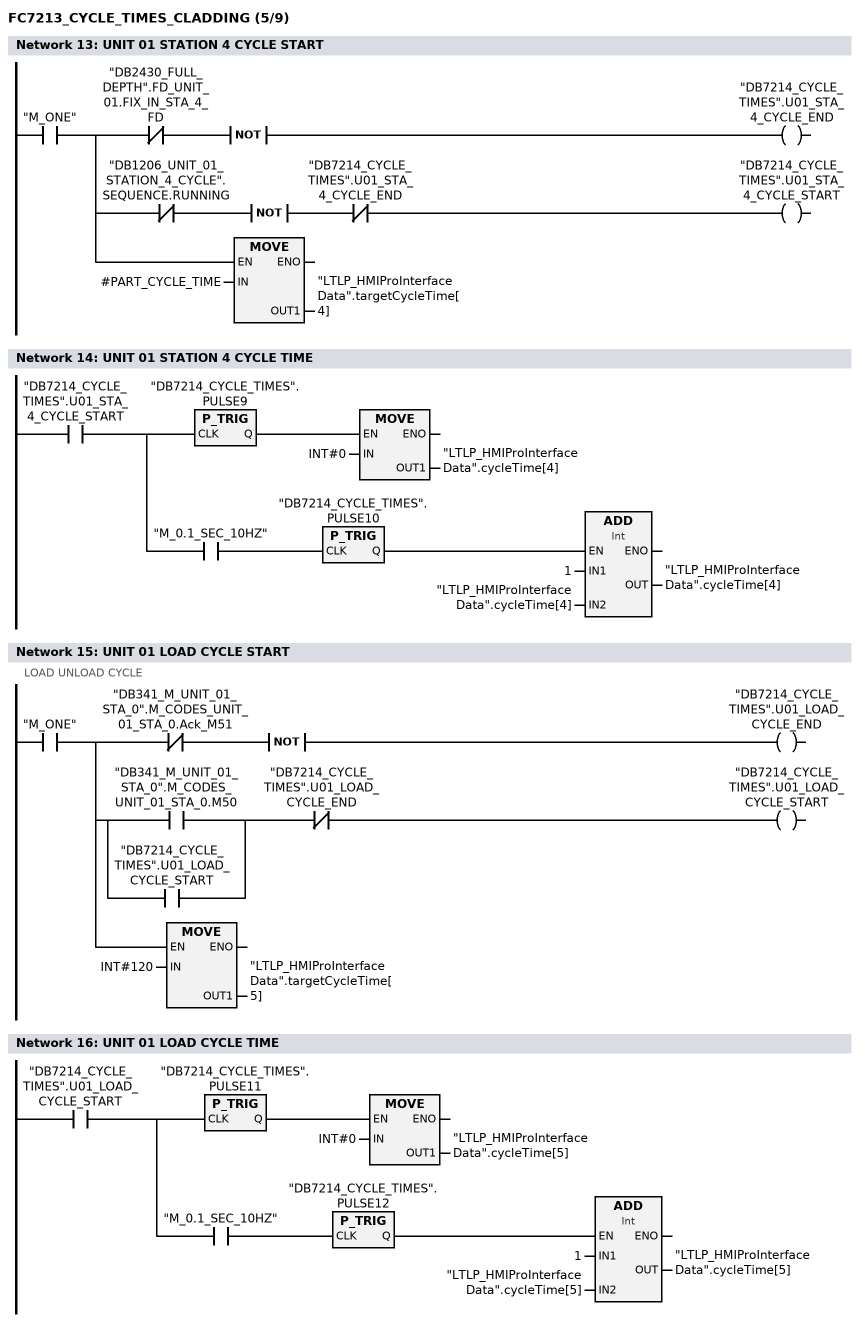
   RUNG wire#powerrail
      Contact( "M_ONE" )
      wire#w1
      I_Contact( "DB2430_FULL_DEPTH".FD_UNIT_01.FIX_IN_STA_4_FD )
      Not()
      Coil( "DB7214_CYCLE_TIMES".U01_STA_4_CYCLE_END )
   END_RUNG
   RUNG wire#w1
      I_Contact( "DB1206_UNIT_01_STATION_4_CYCLE".SEQUENCE.RUNNING )
      Not()
      I_Contact( "DB7214_CYCLE_TIMES".U01_STA_4_CYCLE_END )
      Coil( "DB7214_CYCLE_TIMES".U01_STA_4_CYCLE_START )
   END_RUNG
   RUNG wire#w1
      { S7_GenerateENO := "TRUE" } Move(in := #PART_CYCLE_TIME, out1 => "LTLP_HMIProInterfaceData".targetCycleTime[4])
   END_RUNG
   // the same network as SCL:
   "DB7214_CYCLE_TIMES".U01_STA_4_CYCLE_END := NOT ("M_ONE" AND NOT "DB2430_FULL_DEPTH".FD_UNIT_01.FIX_IN_STA_4_FD);
   "DB7214_CYCLE_TIMES".U01_STA_4_CYCLE_START := NOT ("M_ONE" AND NOT "DB1206_UNIT_01_STATION_4_CYCLE".SEQUENCE.RUNNING) AND NOT "DB7214_CYCLE_TIMES".U01_STA_4_CYCLE_END;
   IF "M_ONE" THEN "LTLP_HMIProInterfaceData".targetCycleTime[4] := #PART_CYCLE_TIME; END_IF;
END_REGION

REGION Network 14: UNIT 01 STATION 4 CYCLE TIME
   RUNG wire#powerrail
      Contact( "DB7214_CYCLE_TIMES".U01_STA_4_CYCLE_START )
      wire#w1
      P_Trig( "DB7214_CYCLE_TIMES".PULSE9 )
      { S7_GenerateENO := "TRUE" } Move(in := INT#0, out1 => "LTLP_HMIProInterfaceData".cycleTime[4])
   END_RUNG
   RUNG wire#w1
      Contact( "M_0.1_SEC_10HZ" )
      P_Trig( "DB7214_CYCLE_TIMES".PULSE10 )
      { S7_Templates := "SrcType := Int"; S7_GenerateENO := "TRUE" } Add(in1 := 1, in2 := "LTLP_HMIProInterfaceData".cycleTime[4], out => "LTLP_HMIProInterfaceData".cycleTime[4])
   END_RUNG
   // the same network as SCL:
   #_w1 := "DB7214_CYCLE_TIMES".U01_STA_4_CYCLE_START AND NOT "DB7214_CYCLE_TIMES".PULSE9;   // rising edge
   "DB7214_CYCLE_TIMES".PULSE9 := "DB7214_CYCLE_TIMES".U01_STA_4_CYCLE_START;
   IF #_w1 THEN "LTLP_HMIProInterfaceData".cycleTime[4] := INT#0; END_IF;
   #_w2 := "DB7214_CYCLE_TIMES".U01_STA_4_CYCLE_START AND "M_0.1_SEC_10HZ";
   #_w3 := #_w2 AND NOT "DB7214_CYCLE_TIMES".PULSE10;   // rising edge
   "DB7214_CYCLE_TIMES".PULSE10 := #_w2;
   IF #_w3 THEN
       "LTLP_HMIProInterfaceData".cycleTime[4] := 1 + "LTLP_HMIProInterfaceData".cycleTime[4];
   END_IF;
END_REGION

REGION Network 15: UNIT 01 LOAD CYCLE START
   // LOAD UNLOAD CYCLE
   RUNG wire#powerrail
      Contact( "M_ONE" )
      wire#w1
      I_Contact( "DB341_M_UNIT_01_STA_0".M_CODES_UNIT_01_STA_0.Ack_M51 )
      Not()
      Coil( "DB7214_CYCLE_TIMES".U01_LOAD_CYCLE_END )
   END_RUNG
   RUNG wire#w1
      Contact( "DB341_M_UNIT_01_STA_0".M_CODES_UNIT_01_STA_0.M50 )
      wire#w2
      I_Contact( "DB7214_CYCLE_TIMES".U01_LOAD_CYCLE_END )
      Coil( "DB7214_CYCLE_TIMES".U01_LOAD_CYCLE_START )
   END_RUNG
   RUNG wire#w1
      Contact( "DB7214_CYCLE_TIMES".U01_LOAD_CYCLE_START )
   END_RUNG wire#w2
   RUNG wire#w1
      { S7_GenerateENO := "TRUE" } Move(in := INT#120, out1 => "LTLP_HMIProInterfaceData".targetCycleTime[5])
   END_RUNG
   // the same network as SCL:
   "DB7214_CYCLE_TIMES".U01_LOAD_CYCLE_END := NOT ("M_ONE" AND NOT "DB341_M_UNIT_01_STA_0".M_CODES_UNIT_01_STA_0.Ack_M51);
   "DB7214_CYCLE_TIMES".U01_LOAD_CYCLE_START := "M_ONE" AND ("DB341_M_UNIT_01_STA_0".M_CODES_UNIT_01_STA_0.M50 OR "DB7214_CYCLE_TIMES".U01_LOAD_CYCLE_START) AND NOT "DB7214_CYCLE_TIMES".U01_LOAD_CYCLE_END;
   IF "M_ONE" THEN "LTLP_HMIProInterfaceData".targetCycleTime[5] := INT#120; END_IF;
END_REGION

REGION Network 16: UNIT 01 LOAD CYCLE TIME
   RUNG wire#powerrail
      Contact( "DB7214_CYCLE_TIMES".U01_LOAD_CYCLE_START )
      wire#w1
      P_Trig( "DB7214_CYCLE_TIMES".PULSE11 )
      { S7_GenerateENO := "TRUE" } Move(in := INT#0, out1 => "LTLP_HMIProInterfaceData".cycleTime[5])
   END_RUNG
   RUNG wire#w1
      Contact( "M_0.1_SEC_10HZ" )
      P_Trig( "DB7214_CYCLE_TIMES".PULSE12 )
      { S7_Templates := "SrcType := Int"; S7_GenerateENO := "TRUE" } Add(in1 := 1, in2 := "LTLP_HMIProInterfaceData".cycleTime[5], out => "LTLP_HMIProInterfaceData".cycleTime[5])
   END_RUNG
   // the same network as SCL:
   #_w1 := "DB7214_CYCLE_TIMES".U01_LOAD_CYCLE_START AND NOT "DB7214_CYCLE_TIMES".PULSE11;   // rising edge
   "DB7214_CYCLE_TIMES".PULSE11 := "DB7214_CYCLE_TIMES".U01_LOAD_CYCLE_START;
   IF #_w1 THEN "LTLP_HMIProInterfaceData".cycleTime[5] := INT#0; END_IF;
   #_w2 := "DB7214_CYCLE_TIMES".U01_LOAD_CYCLE_START AND "M_0.1_SEC_10HZ";
   #_w3 := #_w2 AND NOT "DB7214_CYCLE_TIMES".PULSE12;   // rising edge
   "DB7214_CYCLE_TIMES".PULSE12 := #_w2;
   IF #_w3 THEN
       "LTLP_HMIProInterfaceData".cycleTime[5] := 1 + "LTLP_HMIProInterfaceData".cycleTime[5];
   END_IF;
END_REGION

REGION Network 17: UNIT 02 PART TO PART CYCLE / PART TO PART CYCLE START
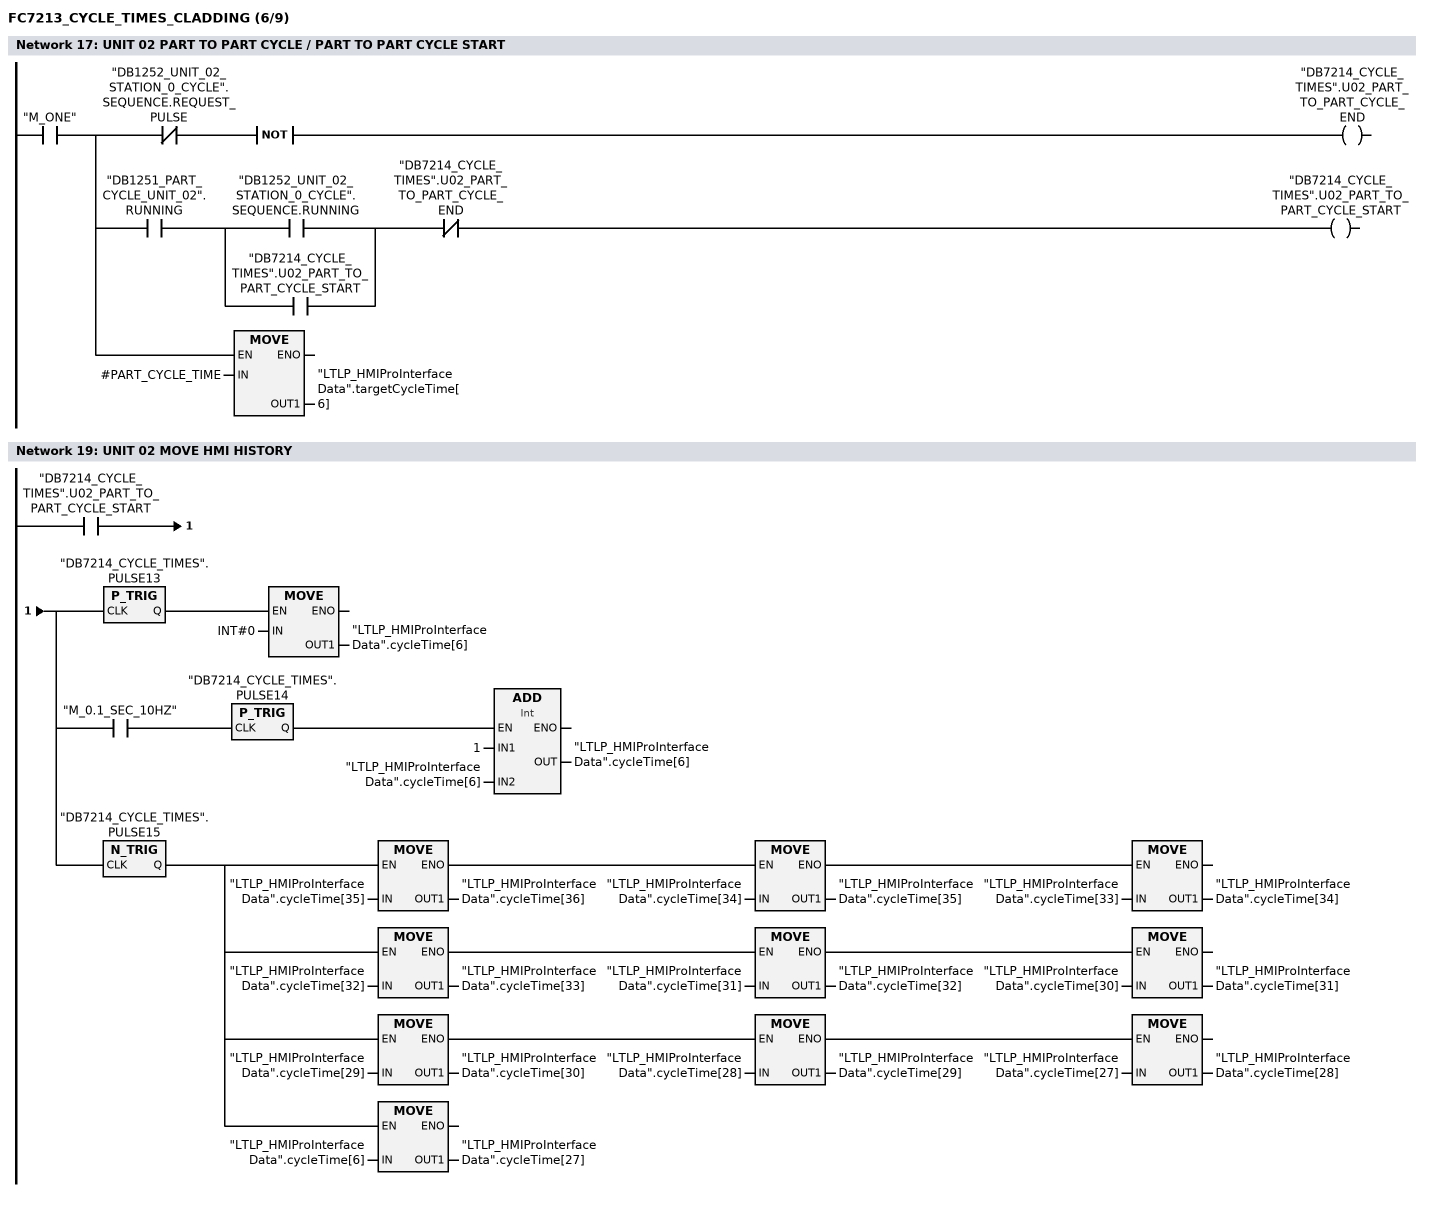
   RUNG wire#powerrail
      Contact( "M_ONE" )
      wire#w1
      I_Contact( "DB1252_UNIT_02_STATION_0_CYCLE".SEQUENCE.REQUEST_PULSE )
      Not()
      Coil( "DB7214_CYCLE_TIMES".U02_PART_TO_PART_CYCLE_END )
   END_RUNG
   RUNG wire#w1
      Contact( "DB1251_PART_CYCLE_UNIT_02".RUNNING )
      wire#w2
      Contact( "DB1252_UNIT_02_STATION_0_CYCLE".SEQUENCE.RUNNING )
      wire#w3
      I_Contact( "DB7214_CYCLE_TIMES".U02_PART_TO_PART_CYCLE_END )
      Coil( "DB7214_CYCLE_TIMES".U02_PART_TO_PART_CYCLE_START )
   END_RUNG
   RUNG wire#w2
      Contact( "DB7214_CYCLE_TIMES".U02_PART_TO_PART_CYCLE_START )
   END_RUNG wire#w3
   RUNG wire#w1
      { S7_GenerateENO := "TRUE" } Move(in := #PART_CYCLE_TIME, out1 => "LTLP_HMIProInterfaceData".targetCycleTime[6])
   END_RUNG
   // the same network as SCL:
   "DB7214_CYCLE_TIMES".U02_PART_TO_PART_CYCLE_END := NOT ("M_ONE" AND NOT "DB1252_UNIT_02_STATION_0_CYCLE".SEQUENCE.REQUEST_PULSE);
   "DB7214_CYCLE_TIMES".U02_PART_TO_PART_CYCLE_START := "M_ONE" AND "DB1251_PART_CYCLE_UNIT_02".RUNNING AND ("DB1252_UNIT_02_STATION_0_CYCLE".SEQUENCE.RUNNING OR "DB7214_CYCLE_TIMES".U02_PART_TO_PART_CYCLE_START) AND NOT "DB7214_CYCLE_TIMES".U02_PART_TO_PART_CYCLE_END;
   IF "M_ONE" THEN "LTLP_HMIProInterfaceData".targetCycleTime[6] := #PART_CYCLE_TIME; END_IF;
END_REGION

NETWORK
TITLE = UNIT 02 HMI HISTORY
      L     "LTLP_HMIProInterfaceData".targetCycleTime[6];
      T     "LTLP_HMIProInterfaceData".targetCycleTime[27];
      T     "LTLP_HMIProInterfaceData".targetCycleTime[28];
      T     "LTLP_HMIProInterfaceData".targetCycleTime[29];
      T     "LTLP_HMIProInterfaceData".targetCycleTime[30];
      T     "LTLP_HMIProInterfaceData".targetCycleTime[31];
      T     "LTLP_HMIProInterfaceData".targetCycleTime[32];
      T     "LTLP_HMIProInterfaceData".targetCycleTime[33];
      T     "LTLP_HMIProInterfaceData".targetCycleTime[34];
      T     "LTLP_HMIProInterfaceData".targetCycleTime[35];
      T     "LTLP_HMIProInterfaceData".targetCycleTime[36];
      NOP   0;

REGION Network 19: UNIT 02 MOVE HMI HISTORY
   RUNG wire#powerrail
      Contact( "DB7214_CYCLE_TIMES".U02_PART_TO_PART_CYCLE_START )
      wire#w1
      P_Trig( "DB7214_CYCLE_TIMES".PULSE13 )
      { S7_GenerateENO := "TRUE" } Move(in := INT#0, out1 => "LTLP_HMIProInterfaceData".cycleTime[6])
   END_RUNG
   RUNG wire#w1
      Contact( "M_0.1_SEC_10HZ" )
      P_Trig( "DB7214_CYCLE_TIMES".PULSE14 )
      { S7_Templates := "SrcType := Int"; S7_GenerateENO := "TRUE" } Add(in1 := 1, in2 := "LTLP_HMIProInterfaceData".cycleTime[6], out => "LTLP_HMIProInterfaceData".cycleTime[6])
   END_RUNG
   RUNG wire#w1
      N_Trig( "DB7214_CYCLE_TIMES".PULSE15 )
      wire#w2
      { S7_GenerateENO := "TRUE" } Move(in := "LTLP_HMIProInterfaceData".cycleTime[35], out1 => "LTLP_HMIProInterfaceData".cycleTime[36])
      { S7_GenerateENO := "TRUE" } Move(in := "LTLP_HMIProInterfaceData".cycleTime[34], out1 => "LTLP_HMIProInterfaceData".cycleTime[35])
      { S7_GenerateENO := "TRUE" } Move(in := "LTLP_HMIProInterfaceData".cycleTime[33], out1 => "LTLP_HMIProInterfaceData".cycleTime[34])
   END_RUNG
   RUNG wire#w2
      { S7_GenerateENO := "TRUE" } Move(in := "LTLP_HMIProInterfaceData".cycleTime[32], out1 => "LTLP_HMIProInterfaceData".cycleTime[33])
      { S7_GenerateENO := "TRUE" } Move(in := "LTLP_HMIProInterfaceData".cycleTime[31], out1 => "LTLP_HMIProInterfaceData".cycleTime[32])
      { S7_GenerateENO := "TRUE" } Move(in := "LTLP_HMIProInterfaceData".cycleTime[30], out1 => "LTLP_HMIProInterfaceData".cycleTime[31])
   END_RUNG
   RUNG wire#w2
      { S7_GenerateENO := "TRUE" } Move(in := "LTLP_HMIProInterfaceData".cycleTime[29], out1 => "LTLP_HMIProInterfaceData".cycleTime[30])
      { S7_GenerateENO := "TRUE" } Move(in := "LTLP_HMIProInterfaceData".cycleTime[28], out1 => "LTLP_HMIProInterfaceData".cycleTime[29])
      { S7_GenerateENO := "TRUE" } Move(in := "LTLP_HMIProInterfaceData".cycleTime[27], out1 => "LTLP_HMIProInterfaceData".cycleTime[28])
   END_RUNG
   RUNG wire#w2
      { S7_GenerateENO := "TRUE" } Move(in := "LTLP_HMIProInterfaceData".cycleTime[6], out1 => "LTLP_HMIProInterfaceData".cycleTime[27])
   END_RUNG
   // the same network as SCL:
   // ENO of a box is taken as its EN; it also drops when the box reports an error
   #_w1 := "DB7214_CYCLE_TIMES".U02_PART_TO_PART_CYCLE_START AND NOT "DB7214_CYCLE_TIMES".PULSE13;   // rising edge
   "DB7214_CYCLE_TIMES".PULSE13 := "DB7214_CYCLE_TIMES".U02_PART_TO_PART_CYCLE_START;
   IF #_w1 THEN "LTLP_HMIProInterfaceData".cycleTime[6] := INT#0; END_IF;
   #_w2 := "DB7214_CYCLE_TIMES".U02_PART_TO_PART_CYCLE_START AND "M_0.1_SEC_10HZ";
   #_w3 := #_w2 AND NOT "DB7214_CYCLE_TIMES".PULSE14;   // rising edge
   "DB7214_CYCLE_TIMES".PULSE14 := #_w2;
   IF #_w3 THEN
       "LTLP_HMIProInterfaceData".cycleTime[6] := 1 + "LTLP_HMIProInterfaceData".cycleTime[6];
   END_IF;
   #_w4 := NOT "DB7214_CYCLE_TIMES".U02_PART_TO_PART_CYCLE_START AND "DB7214_CYCLE_TIMES".PULSE15;   // falling edge
   "DB7214_CYCLE_TIMES".PULSE15 := "DB7214_CYCLE_TIMES".U02_PART_TO_PART_CYCLE_START;
   IF #_w4 THEN
       "LTLP_HMIProInterfaceData".cycleTime[36] := "LTLP_HMIProInterfaceData".cycleTime[35];
       "LTLP_HMIProInterfaceData".cycleTime[35] := "LTLP_HMIProInterfaceData".cycleTime[34];
       "LTLP_HMIProInterfaceData".cycleTime[34] := "LTLP_HMIProInterfaceData".cycleTime[33];
       "LTLP_HMIProInterfaceData".cycleTime[33] := "LTLP_HMIProInterfaceData".cycleTime[32];
       "LTLP_HMIProInterfaceData".cycleTime[32] := "LTLP_HMIProInterfaceData".cycleTime[31];
       "LTLP_HMIProInterfaceData".cycleTime[31] := "LTLP_HMIProInterfaceData".cycleTime[30];
       "LTLP_HMIProInterfaceData".cycleTime[30] := "LTLP_HMIProInterfaceData".cycleTime[29];
       "LTLP_HMIProInterfaceData".cycleTime[29] := "LTLP_HMIProInterfaceData".cycleTime[28];
       "LTLP_HMIProInterfaceData".cycleTime[28] := "LTLP_HMIProInterfaceData".cycleTime[27];
       "LTLP_HMIProInterfaceData".cycleTime[27] := "LTLP_HMIProInterfaceData".cycleTime[6];
   END_IF;
END_REGION

REGION Network 20: UNIT 02 STATION 1 CYCLE START
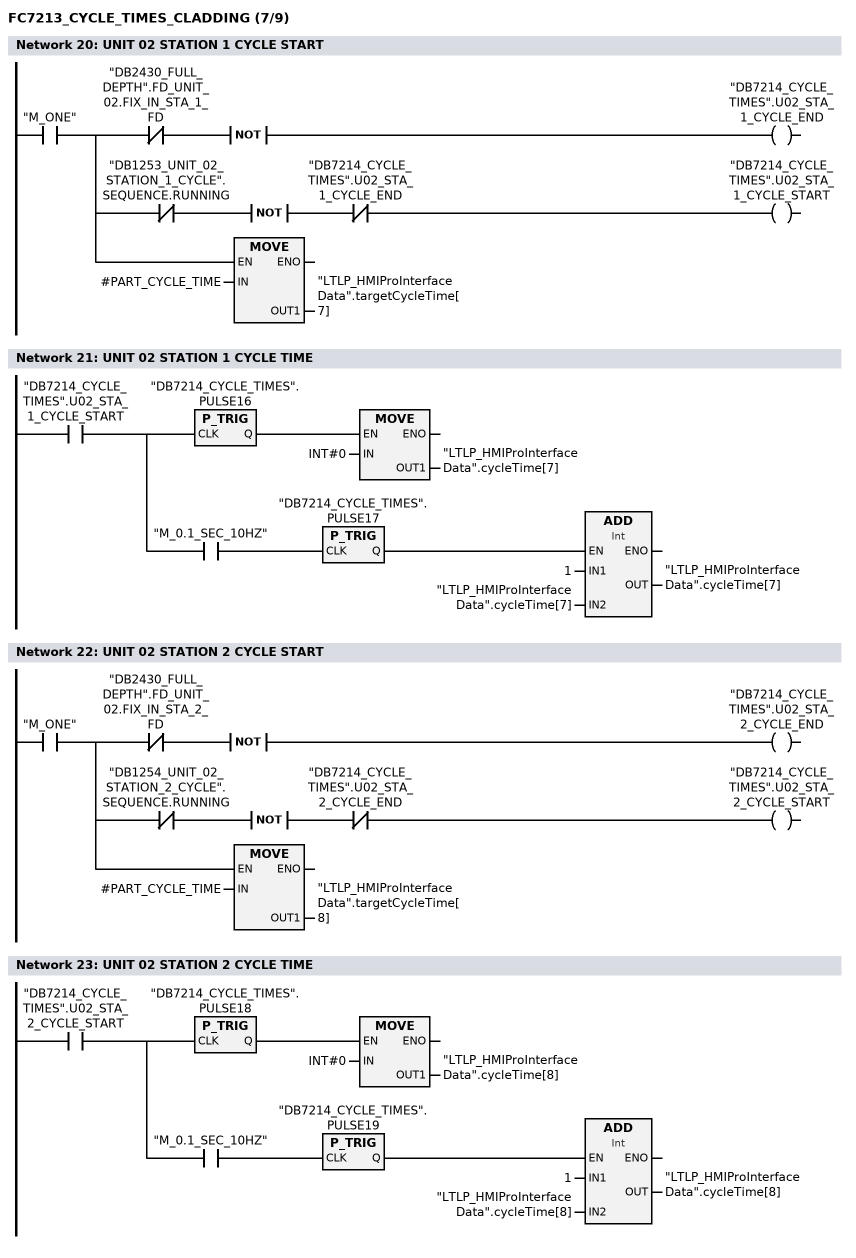
   RUNG wire#powerrail
      Contact( "M_ONE" )
      wire#w1
      I_Contact( "DB2430_FULL_DEPTH".FD_UNIT_02.FIX_IN_STA_1_FD )
      Not()
      Coil( "DB7214_CYCLE_TIMES".U02_STA_1_CYCLE_END )
   END_RUNG
   RUNG wire#w1
      I_Contact( "DB1253_UNIT_02_STATION_1_CYCLE".SEQUENCE.RUNNING )
      Not()
      I_Contact( "DB7214_CYCLE_TIMES".U02_STA_1_CYCLE_END )
      Coil( "DB7214_CYCLE_TIMES".U02_STA_1_CYCLE_START )
   END_RUNG
   RUNG wire#w1
      { S7_GenerateENO := "TRUE" } Move(in := #PART_CYCLE_TIME, out1 => "LTLP_HMIProInterfaceData".targetCycleTime[7])
   END_RUNG
   // the same network as SCL:
   "DB7214_CYCLE_TIMES".U02_STA_1_CYCLE_END := NOT ("M_ONE" AND NOT "DB2430_FULL_DEPTH".FD_UNIT_02.FIX_IN_STA_1_FD);
   "DB7214_CYCLE_TIMES".U02_STA_1_CYCLE_START := NOT ("M_ONE" AND NOT "DB1253_UNIT_02_STATION_1_CYCLE".SEQUENCE.RUNNING) AND NOT "DB7214_CYCLE_TIMES".U02_STA_1_CYCLE_END;
   IF "M_ONE" THEN "LTLP_HMIProInterfaceData".targetCycleTime[7] := #PART_CYCLE_TIME; END_IF;
END_REGION

REGION Network 21: UNIT 02 STATION 1 CYCLE TIME
   RUNG wire#powerrail
      Contact( "DB7214_CYCLE_TIMES".U02_STA_1_CYCLE_START )
      wire#w1
      P_Trig( "DB7214_CYCLE_TIMES".PULSE16 )
      { S7_GenerateENO := "TRUE" } Move(in := INT#0, out1 => "LTLP_HMIProInterfaceData".cycleTime[7])
   END_RUNG
   RUNG wire#w1
      Contact( "M_0.1_SEC_10HZ" )
      P_Trig( "DB7214_CYCLE_TIMES".PULSE17 )
      { S7_Templates := "SrcType := Int"; S7_GenerateENO := "TRUE" } Add(in1 := 1, in2 := "LTLP_HMIProInterfaceData".cycleTime[7], out => "LTLP_HMIProInterfaceData".cycleTime[7])
   END_RUNG
   // the same network as SCL:
   #_w1 := "DB7214_CYCLE_TIMES".U02_STA_1_CYCLE_START AND NOT "DB7214_CYCLE_TIMES".PULSE16;   // rising edge
   "DB7214_CYCLE_TIMES".PULSE16 := "DB7214_CYCLE_TIMES".U02_STA_1_CYCLE_START;
   IF #_w1 THEN "LTLP_HMIProInterfaceData".cycleTime[7] := INT#0; END_IF;
   #_w2 := "DB7214_CYCLE_TIMES".U02_STA_1_CYCLE_START AND "M_0.1_SEC_10HZ";
   #_w3 := #_w2 AND NOT "DB7214_CYCLE_TIMES".PULSE17;   // rising edge
   "DB7214_CYCLE_TIMES".PULSE17 := #_w2;
   IF #_w3 THEN
       "LTLP_HMIProInterfaceData".cycleTime[7] := 1 + "LTLP_HMIProInterfaceData".cycleTime[7];
   END_IF;
END_REGION

REGION Network 22: UNIT 02 STATION 2 CYCLE START
   RUNG wire#powerrail
      Contact( "M_ONE" )
      wire#w1
      I_Contact( "DB2430_FULL_DEPTH".FD_UNIT_02.FIX_IN_STA_2_FD )
      Not()
      Coil( "DB7214_CYCLE_TIMES".U02_STA_2_CYCLE_END )
   END_RUNG
   RUNG wire#w1
      I_Contact( "DB1254_UNIT_02_STATION_2_CYCLE".SEQUENCE.RUNNING )
      Not()
      I_Contact( "DB7214_CYCLE_TIMES".U02_STA_2_CYCLE_END )
      Coil( "DB7214_CYCLE_TIMES".U02_STA_2_CYCLE_START )
   END_RUNG
   RUNG wire#w1
      { S7_GenerateENO := "TRUE" } Move(in := #PART_CYCLE_TIME, out1 => "LTLP_HMIProInterfaceData".targetCycleTime[8])
   END_RUNG
   // the same network as SCL:
   "DB7214_CYCLE_TIMES".U02_STA_2_CYCLE_END := NOT ("M_ONE" AND NOT "DB2430_FULL_DEPTH".FD_UNIT_02.FIX_IN_STA_2_FD);
   "DB7214_CYCLE_TIMES".U02_STA_2_CYCLE_START := NOT ("M_ONE" AND NOT "DB1254_UNIT_02_STATION_2_CYCLE".SEQUENCE.RUNNING) AND NOT "DB7214_CYCLE_TIMES".U02_STA_2_CYCLE_END;
   IF "M_ONE" THEN "LTLP_HMIProInterfaceData".targetCycleTime[8] := #PART_CYCLE_TIME; END_IF;
END_REGION

REGION Network 23: UNIT 02 STATION 2 CYCLE TIME
   RUNG wire#powerrail
      Contact( "DB7214_CYCLE_TIMES".U02_STA_2_CYCLE_START )
      wire#w1
      P_Trig( "DB7214_CYCLE_TIMES".PULSE18 )
      { S7_GenerateENO := "TRUE" } Move(in := INT#0, out1 => "LTLP_HMIProInterfaceData".cycleTime[8])
   END_RUNG
   RUNG wire#w1
      Contact( "M_0.1_SEC_10HZ" )
      P_Trig( "DB7214_CYCLE_TIMES".PULSE19 )
      { S7_Templates := "SrcType := Int"; S7_GenerateENO := "TRUE" } Add(in1 := 1, in2 := "LTLP_HMIProInterfaceData".cycleTime[8], out => "LTLP_HMIProInterfaceData".cycleTime[8])
   END_RUNG
   // the same network as SCL:
   #_w1 := "DB7214_CYCLE_TIMES".U02_STA_2_CYCLE_START AND NOT "DB7214_CYCLE_TIMES".PULSE18;   // rising edge
   "DB7214_CYCLE_TIMES".PULSE18 := "DB7214_CYCLE_TIMES".U02_STA_2_CYCLE_START;
   IF #_w1 THEN "LTLP_HMIProInterfaceData".cycleTime[8] := INT#0; END_IF;
   #_w2 := "DB7214_CYCLE_TIMES".U02_STA_2_CYCLE_START AND "M_0.1_SEC_10HZ";
   #_w3 := #_w2 AND NOT "DB7214_CYCLE_TIMES".PULSE19;   // rising edge
   "DB7214_CYCLE_TIMES".PULSE19 := #_w2;
   IF #_w3 THEN
       "LTLP_HMIProInterfaceData".cycleTime[8] := 1 + "LTLP_HMIProInterfaceData".cycleTime[8];
   END_IF;
END_REGION

REGION Network 24: UNIT 02 STATION 3 CYCLE START
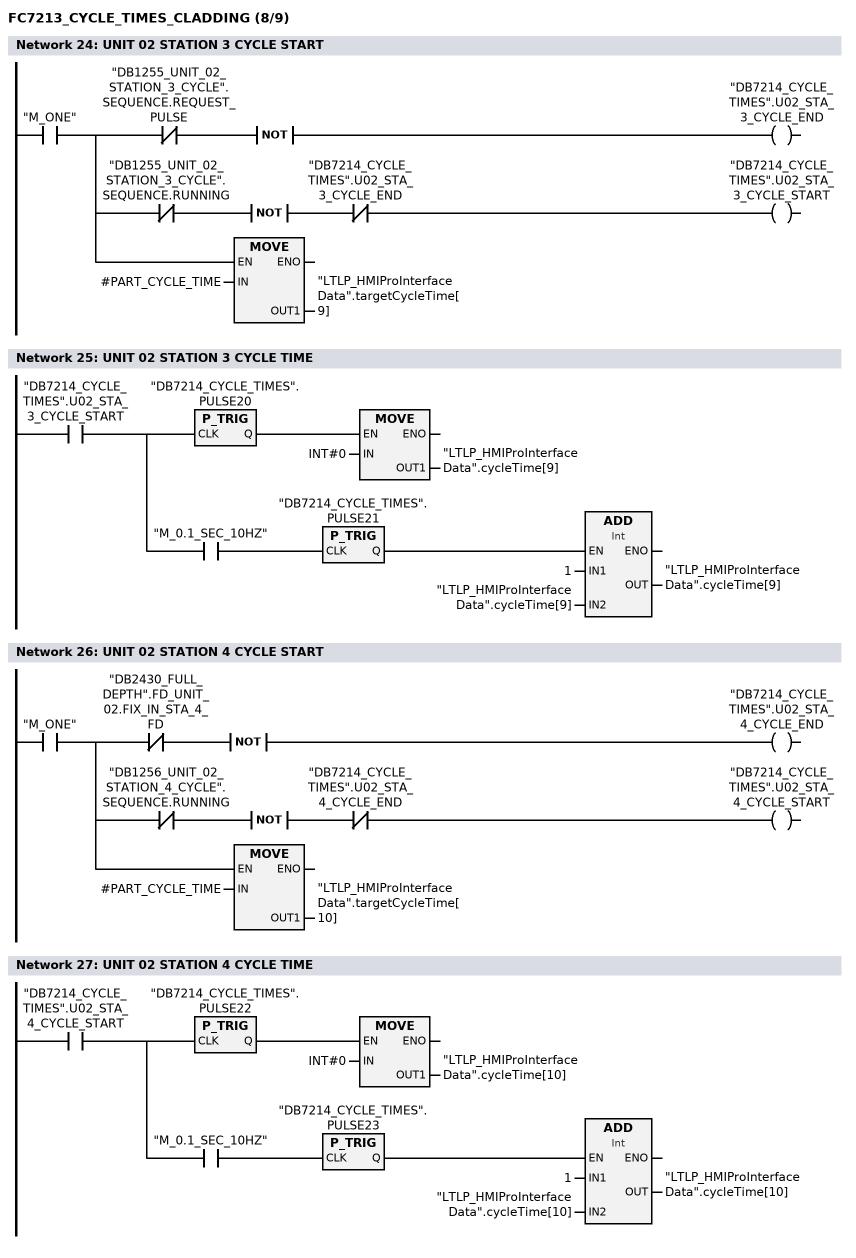
   RUNG wire#powerrail
      Contact( "M_ONE" )
      wire#w1
      I_Contact( "DB1255_UNIT_02_STATION_3_CYCLE".SEQUENCE.REQUEST_PULSE )
      Not()
      Coil( "DB7214_CYCLE_TIMES".U02_STA_3_CYCLE_END )
   END_RUNG
   RUNG wire#w1
      I_Contact( "DB1255_UNIT_02_STATION_3_CYCLE".SEQUENCE.RUNNING )
      Not()
      I_Contact( "DB7214_CYCLE_TIMES".U02_STA_3_CYCLE_END )
      Coil( "DB7214_CYCLE_TIMES".U02_STA_3_CYCLE_START )
   END_RUNG
   RUNG wire#w1
      { S7_GenerateENO := "TRUE" } Move(in := #PART_CYCLE_TIME, out1 => "LTLP_HMIProInterfaceData".targetCycleTime[9])
   END_RUNG
   // the same network as SCL:
   "DB7214_CYCLE_TIMES".U02_STA_3_CYCLE_END := NOT ("M_ONE" AND NOT "DB1255_UNIT_02_STATION_3_CYCLE".SEQUENCE.REQUEST_PULSE);
   "DB7214_CYCLE_TIMES".U02_STA_3_CYCLE_START := NOT ("M_ONE" AND NOT "DB1255_UNIT_02_STATION_3_CYCLE".SEQUENCE.RUNNING) AND NOT "DB7214_CYCLE_TIMES".U02_STA_3_CYCLE_END;
   IF "M_ONE" THEN "LTLP_HMIProInterfaceData".targetCycleTime[9] := #PART_CYCLE_TIME; END_IF;
END_REGION

REGION Network 25: UNIT 02 STATION 3 CYCLE TIME
   RUNG wire#powerrail
      Contact( "DB7214_CYCLE_TIMES".U02_STA_3_CYCLE_START )
      wire#w1
      P_Trig( "DB7214_CYCLE_TIMES".PULSE20 )
      { S7_GenerateENO := "TRUE" } Move(in := INT#0, out1 => "LTLP_HMIProInterfaceData".cycleTime[9])
   END_RUNG
   RUNG wire#w1
      Contact( "M_0.1_SEC_10HZ" )
      P_Trig( "DB7214_CYCLE_TIMES".PULSE21 )
      { S7_Templates := "SrcType := Int"; S7_GenerateENO := "TRUE" } Add(in1 := 1, in2 := "LTLP_HMIProInterfaceData".cycleTime[9], out => "LTLP_HMIProInterfaceData".cycleTime[9])
   END_RUNG
   // the same network as SCL:
   #_w1 := "DB7214_CYCLE_TIMES".U02_STA_3_CYCLE_START AND NOT "DB7214_CYCLE_TIMES".PULSE20;   // rising edge
   "DB7214_CYCLE_TIMES".PULSE20 := "DB7214_CYCLE_TIMES".U02_STA_3_CYCLE_START;
   IF #_w1 THEN "LTLP_HMIProInterfaceData".cycleTime[9] := INT#0; END_IF;
   #_w2 := "DB7214_CYCLE_TIMES".U02_STA_3_CYCLE_START AND "M_0.1_SEC_10HZ";
   #_w3 := #_w2 AND NOT "DB7214_CYCLE_TIMES".PULSE21;   // rising edge
   "DB7214_CYCLE_TIMES".PULSE21 := #_w2;
   IF #_w3 THEN
       "LTLP_HMIProInterfaceData".cycleTime[9] := 1 + "LTLP_HMIProInterfaceData".cycleTime[9];
   END_IF;
END_REGION

REGION Network 26: UNIT 02 STATION 4 CYCLE START
   RUNG wire#powerrail
      Contact( "M_ONE" )
      wire#w1
      I_Contact( "DB2430_FULL_DEPTH".FD_UNIT_02.FIX_IN_STA_4_FD )
      Not()
      Coil( "DB7214_CYCLE_TIMES".U02_STA_4_CYCLE_END )
   END_RUNG
   RUNG wire#w1
      I_Contact( "DB1256_UNIT_02_STATION_4_CYCLE".SEQUENCE.RUNNING )
      Not()
      I_Contact( "DB7214_CYCLE_TIMES".U02_STA_4_CYCLE_END )
      Coil( "DB7214_CYCLE_TIMES".U02_STA_4_CYCLE_START )
   END_RUNG
   RUNG wire#w1
      { S7_GenerateENO := "TRUE" } Move(in := #PART_CYCLE_TIME, out1 => "LTLP_HMIProInterfaceData".targetCycleTime[10])
   END_RUNG
   // the same network as SCL:
   "DB7214_CYCLE_TIMES".U02_STA_4_CYCLE_END := NOT ("M_ONE" AND NOT "DB2430_FULL_DEPTH".FD_UNIT_02.FIX_IN_STA_4_FD);
   "DB7214_CYCLE_TIMES".U02_STA_4_CYCLE_START := NOT ("M_ONE" AND NOT "DB1256_UNIT_02_STATION_4_CYCLE".SEQUENCE.RUNNING) AND NOT "DB7214_CYCLE_TIMES".U02_STA_4_CYCLE_END;
   IF "M_ONE" THEN "LTLP_HMIProInterfaceData".targetCycleTime[10] := #PART_CYCLE_TIME; END_IF;
END_REGION

REGION Network 27: UNIT 02 STATION 4 CYCLE TIME
   RUNG wire#powerrail
      Contact( "DB7214_CYCLE_TIMES".U02_STA_4_CYCLE_START )
      wire#w1
      P_Trig( "DB7214_CYCLE_TIMES".PULSE22 )
      { S7_GenerateENO := "TRUE" } Move(in := INT#0, out1 => "LTLP_HMIProInterfaceData".cycleTime[10])
   END_RUNG
   RUNG wire#w1
      Contact( "M_0.1_SEC_10HZ" )
      P_Trig( "DB7214_CYCLE_TIMES".PULSE23 )
      { S7_Templates := "SrcType := Int"; S7_GenerateENO := "TRUE" } Add(in1 := 1, in2 := "LTLP_HMIProInterfaceData".cycleTime[10], out => "LTLP_HMIProInterfaceData".cycleTime[10])
   END_RUNG
   // the same network as SCL:
   #_w1 := "DB7214_CYCLE_TIMES".U02_STA_4_CYCLE_START AND NOT "DB7214_CYCLE_TIMES".PULSE22;   // rising edge
   "DB7214_CYCLE_TIMES".PULSE22 := "DB7214_CYCLE_TIMES".U02_STA_4_CYCLE_START;
   IF #_w1 THEN "LTLP_HMIProInterfaceData".cycleTime[10] := INT#0; END_IF;
   #_w2 := "DB7214_CYCLE_TIMES".U02_STA_4_CYCLE_START AND "M_0.1_SEC_10HZ";
   #_w3 := #_w2 AND NOT "DB7214_CYCLE_TIMES".PULSE23;   // rising edge
   "DB7214_CYCLE_TIMES".PULSE23 := #_w2;
   IF #_w3 THEN
       "LTLP_HMIProInterfaceData".cycleTime[10] := 1 + "LTLP_HMIProInterfaceData".cycleTime[10];
   END_IF;
END_REGION

REGION Network 28: UNIT 02 LOAD CYCLE START
   // LOAD UNLOAD CYCLE
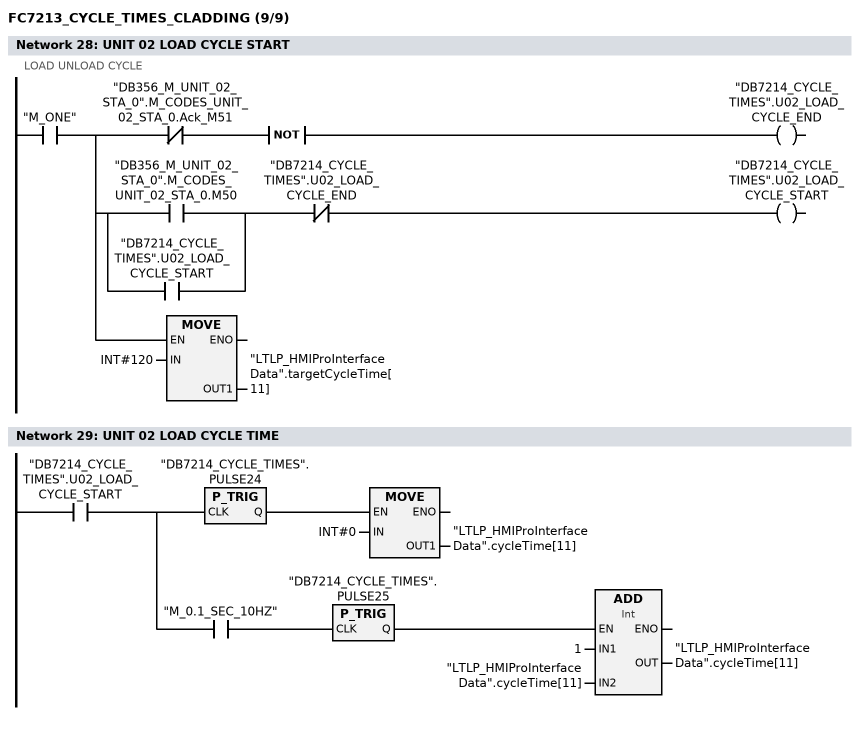
   RUNG wire#powerrail
      Contact( "M_ONE" )
      wire#w1
      I_Contact( "DB356_M_UNIT_02_STA_0".M_CODES_UNIT_02_STA_0.Ack_M51 )
      Not()
      Coil( "DB7214_CYCLE_TIMES".U02_LOAD_CYCLE_END )
   END_RUNG
   RUNG wire#w1
      Contact( "DB356_M_UNIT_02_STA_0".M_CODES_UNIT_02_STA_0.M50 )
      wire#w2
      I_Contact( "DB7214_CYCLE_TIMES".U02_LOAD_CYCLE_END )
      Coil( "DB7214_CYCLE_TIMES".U02_LOAD_CYCLE_START )
   END_RUNG
   RUNG wire#w1
      Contact( "DB7214_CYCLE_TIMES".U02_LOAD_CYCLE_START )
   END_RUNG wire#w2
   RUNG wire#w1
      { S7_GenerateENO := "TRUE" } Move(in := INT#120, out1 => "LTLP_HMIProInterfaceData".targetCycleTime[11])
   END_RUNG
   // the same network as SCL:
   "DB7214_CYCLE_TIMES".U02_LOAD_CYCLE_END := NOT ("M_ONE" AND NOT "DB356_M_UNIT_02_STA_0".M_CODES_UNIT_02_STA_0.Ack_M51);
   "DB7214_CYCLE_TIMES".U02_LOAD_CYCLE_START := "M_ONE" AND ("DB356_M_UNIT_02_STA_0".M_CODES_UNIT_02_STA_0.M50 OR "DB7214_CYCLE_TIMES".U02_LOAD_CYCLE_START) AND NOT "DB7214_CYCLE_TIMES".U02_LOAD_CYCLE_END;
   IF "M_ONE" THEN "LTLP_HMIProInterfaceData".targetCycleTime[11] := INT#120; END_IF;
END_REGION

REGION Network 29: UNIT 02 LOAD CYCLE TIME
   RUNG wire#powerrail
      Contact( "DB7214_CYCLE_TIMES".U02_LOAD_CYCLE_START )
      wire#w1
      P_Trig( "DB7214_CYCLE_TIMES".PULSE24 )
      { S7_GenerateENO := "TRUE" } Move(in := INT#0, out1 => "LTLP_HMIProInterfaceData".cycleTime[11])
   END_RUNG
   RUNG wire#w1
      Contact( "M_0.1_SEC_10HZ" )
      P_Trig( "DB7214_CYCLE_TIMES".PULSE25 )
      { S7_Templates := "SrcType := Int"; S7_GenerateENO := "TRUE" } Add(in1 := 1, in2 := "LTLP_HMIProInterfaceData".cycleTime[11], out => "LTLP_HMIProInterfaceData".cycleTime[11])
   END_RUNG
   // the same network as SCL:
   #_w1 := "DB7214_CYCLE_TIMES".U02_LOAD_CYCLE_START AND NOT "DB7214_CYCLE_TIMES".PULSE24;   // rising edge
   "DB7214_CYCLE_TIMES".PULSE24 := "DB7214_CYCLE_TIMES".U02_LOAD_CYCLE_START;
   IF #_w1 THEN "LTLP_HMIProInterfaceData".cycleTime[11] := INT#0; END_IF;
   #_w2 := "DB7214_CYCLE_TIMES".U02_LOAD_CYCLE_START AND "M_0.1_SEC_10HZ";
   #_w3 := #_w2 AND NOT "DB7214_CYCLE_TIMES".PULSE25;   // rising edge
   "DB7214_CYCLE_TIMES".PULSE25 := #_w2;
   IF #_w3 THEN
       "LTLP_HMIProInterfaceData".cycleTime[11] := 1 + "LTLP_HMIProInterfaceData".cycleTime[11];
   END_IF;
END_REGION
END_FUNCTION
